Staubli VAL3: FC_EndMotion.pgx

program FC_EndMotion()
begin
  //this function is to finish the sychronous motion
  $movejSyncEnd()
end
